// TIA Portal V18 export
// export: Created 2026-04-18T00:00:00Z, ExportSetting WithDefaults
ORGANIZATION_BLOCK "OB31_PID_PLC2_Bon4"   // OB31, LAD, CyclicInterrupt
{ S7_Optimized_Access := 'TRUE' }
VERSION : 0.1
// stored: AutoNumber true, IsIECCheckEnabled false
   VAR_INPUT
      Initial_Call : Bool;
      Remanence : Bool;
   END_VAR
BEGIN

REGION Network 1: Initialize PID Bon 4 Kp parameter
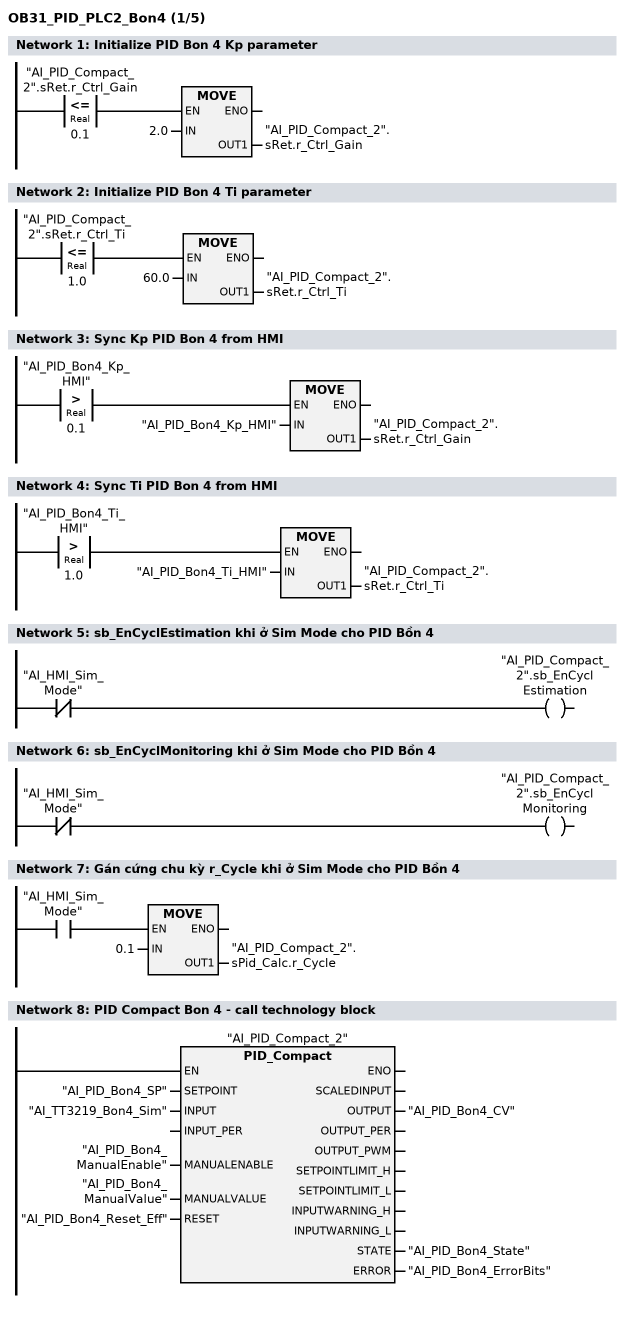
   RUNG wire#powerrail
      { S7_Templates := "SrcType := Real" } LE_Contact(in1 := "AI_PID_Compact_2".sRet.r_Ctrl_Gain, in2 := 0.1)
      { S7_GenerateENO := "TRUE" } Move(in := 2.0, out1 => "AI_PID_Compact_2".sRet.r_Ctrl_Gain)
   END_RUNG
   // the same network as SCL:
   IF "AI_PID_Compact_2".sRet.r_Ctrl_Gain <= 0.1 THEN "AI_PID_Compact_2".sRet.r_Ctrl_Gain := 2.0; END_IF;
END_REGION

REGION Network 2: Initialize PID Bon 4 Ti parameter
   RUNG wire#powerrail
      { S7_Templates := "SrcType := Real" } LE_Contact(in1 := "AI_PID_Compact_2".sRet.r_Ctrl_Ti, in2 := 1.0)
      { S7_GenerateENO := "TRUE" } Move(in := 60.0, out1 => "AI_PID_Compact_2".sRet.r_Ctrl_Ti)
   END_RUNG
   // the same network as SCL:
   IF "AI_PID_Compact_2".sRet.r_Ctrl_Ti <= 1.0 THEN "AI_PID_Compact_2".sRet.r_Ctrl_Ti := 60.0; END_IF;
END_REGION

REGION Network 3: Sync Kp PID Bon 4 from HMI
   RUNG wire#powerrail
      { S7_Templates := "SrcType := Real" } GT_Contact(in1 := "AI_PID_Bon4_Kp_HMI", in2 := 0.1)
      { S7_GenerateENO := "TRUE" } Move(in := "AI_PID_Bon4_Kp_HMI", out1 => "AI_PID_Compact_2".sRet.r_Ctrl_Gain)
   END_RUNG
   // the same network as SCL:
   IF "AI_PID_Bon4_Kp_HMI" > 0.1 THEN "AI_PID_Compact_2".sRet.r_Ctrl_Gain := "AI_PID_Bon4_Kp_HMI"; END_IF;
END_REGION

REGION Network 4: Sync Ti PID Bon 4 from HMI
   RUNG wire#powerrail
      { S7_Templates := "SrcType := Real" } GT_Contact(in1 := "AI_PID_Bon4_Ti_HMI", in2 := 1.0)
      { S7_GenerateENO := "TRUE" } Move(in := "AI_PID_Bon4_Ti_HMI", out1 => "AI_PID_Compact_2".sRet.r_Ctrl_Ti)
   END_RUNG
   // the same network as SCL:
   IF "AI_PID_Bon4_Ti_HMI" > 1.0 THEN "AI_PID_Compact_2".sRet.r_Ctrl_Ti := "AI_PID_Bon4_Ti_HMI"; END_IF;
END_REGION

REGION Network 5: sb_EnCyclEstimation khi ở Sim Mode cho PID Bồn 4
   RUNG wire#powerrail
      I_Contact( "AI_HMI_Sim_Mode" )
      Coil( "AI_PID_Compact_2".sb_EnCyclEstimation )
   END_RUNG
   // the same network as SCL:
   "AI_PID_Compact_2".sb_EnCyclEstimation := NOT "AI_HMI_Sim_Mode";
END_REGION

REGION Network 6: sb_EnCyclMonitoring khi ở Sim Mode cho PID Bồn 4
   RUNG wire#powerrail
      I_Contact( "AI_HMI_Sim_Mode" )
      Coil( "AI_PID_Compact_2".sb_EnCyclMonitoring )
   END_RUNG
   // the same network as SCL:
   "AI_PID_Compact_2".sb_EnCyclMonitoring := NOT "AI_HMI_Sim_Mode";
END_REGION

REGION Network 7: Gán cứng chu kỳ r_Cycle khi ở Sim Mode cho PID Bồn 4
   RUNG wire#powerrail
      Contact( "AI_HMI_Sim_Mode" )
      { S7_GenerateENO := "TRUE" } Move(in := 0.1, out1 => "AI_PID_Compact_2".sPid_Calc.r_Cycle)
   END_RUNG
   // the same network as SCL:
   IF "AI_HMI_Sim_Mode" THEN "AI_PID_Compact_2".sPid_Calc.r_Cycle := 0.1; END_IF;
END_REGION

REGION Network 8: PID Compact Bon 4 - call technology block
   RUNG wire#powerrail
      "AI_PID_Compact_2".PID_Compact(Setpoint := "AI_PID_Bon4_SP", Input := "AI_TT3219_Bon4_Sim", Input_PER :=, ManualEnable := "AI_PID_Bon4_ManualEnable", ManualValue := "AI_PID_Bon4_ManualValue", Reset := "AI_PID_Bon4_Reset_Eff", ScaledInput =>, Output => "AI_PID_Bon4_CV", Output_PER =>, Output_PWM =>, SetpointLimit_H =>, SetpointLimit_L =>, InputWarning_H =>, InputWarning_L =>, State => "AI_PID_Bon4_State", Error => "AI_PID_Bon4_ErrorBits")
   END_RUNG
   // the same network as SCL:
   "AI_PID_Compact_2"(Setpoint := "AI_PID_Bon4_SP",   // PID_Compact
                      Input := "AI_TT3219_Bon4_Sim",
                      ManualEnable := "AI_PID_Bon4_ManualEnable",
                      ManualValue := "AI_PID_Bon4_ManualValue",
                      Reset := "AI_PID_Bon4_Reset_Eff",
                      Output => "AI_PID_Bon4_CV",
                      State => "AI_PID_Bon4_State",
                      Error => "AI_PID_Bon4_ErrorBits");
END_REGION

REGION Network 9: Detect PID Bon 4 Error
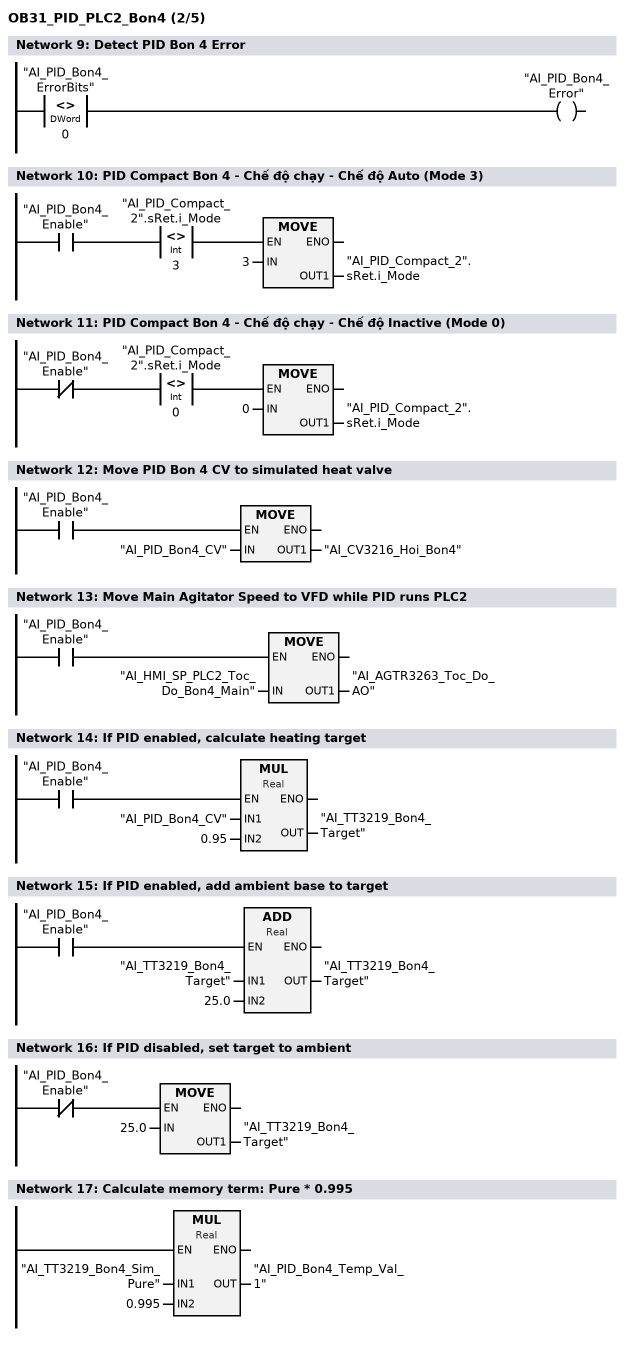
   RUNG wire#powerrail
      { S7_Templates := "SrcType := DWord" } NE_Contact(in1 := "AI_PID_Bon4_ErrorBits", in2 := 0)
      Coil( "AI_PID_Bon4_Error" )
   END_RUNG
   // the same network as SCL:
   "AI_PID_Bon4_Error" := "AI_PID_Bon4_ErrorBits" <> 0;
END_REGION

REGION Network 10: PID Compact Bon 4 - Chế độ chạy - Chế độ Auto (Mode 3)
   RUNG wire#powerrail
      Contact( "AI_PID_Bon4_Enable" )
      { S7_Templates := "SrcType := Int" } NE_Contact(in1 := "AI_PID_Compact_2".sRet.i_Mode, in2 := 3)
      { S7_GenerateENO := "TRUE" } Move(in := 3, out1 => "AI_PID_Compact_2".sRet.i_Mode)
   END_RUNG
   // the same network as SCL:
   IF "AI_PID_Bon4_Enable" AND ("AI_PID_Compact_2".sRet.i_Mode <> 3) THEN
       "AI_PID_Compact_2".sRet.i_Mode := 3;
   END_IF;
END_REGION

REGION Network 11: PID Compact Bon 4 - Chế độ chạy - Chế độ Inactive (Mode 0)
   RUNG wire#powerrail
      I_Contact( "AI_PID_Bon4_Enable" )
      { S7_Templates := "SrcType := Int" } NE_Contact(in1 := "AI_PID_Compact_2".sRet.i_Mode, in2 := 0)
      { S7_GenerateENO := "TRUE" } Move(in := 0, out1 => "AI_PID_Compact_2".sRet.i_Mode)
   END_RUNG
   // the same network as SCL:
   IF NOT "AI_PID_Bon4_Enable" AND ("AI_PID_Compact_2".sRet.i_Mode <> 0) THEN
       "AI_PID_Compact_2".sRet.i_Mode := 0;
   END_IF;
END_REGION

REGION Network 12: Move PID Bon 4 CV to simulated heat valve
   RUNG wire#powerrail
      Contact( "AI_PID_Bon4_Enable" )
      { S7_GenerateENO := "TRUE" } Move(in := "AI_PID_Bon4_CV", out1 => "AI_CV3216_Hoi_Bon4")
   END_RUNG
   // the same network as SCL:
   IF "AI_PID_Bon4_Enable" THEN "AI_CV3216_Hoi_Bon4" := "AI_PID_Bon4_CV"; END_IF;
END_REGION

REGION Network 13: Move Main Agitator Speed to VFD while PID runs PLC2
   RUNG wire#powerrail
      Contact( "AI_PID_Bon4_Enable" )
      { S7_GenerateENO := "TRUE" } Move(in := "AI_HMI_SP_PLC2_Toc_Do_Bon4_Main", out1 => "AI_AGTR3263_Toc_Do_AO")
   END_RUNG
   // the same network as SCL:
   IF "AI_PID_Bon4_Enable" THEN "AI_AGTR3263_Toc_Do_AO" := "AI_HMI_SP_PLC2_Toc_Do_Bon4_Main"; END_IF;
END_REGION

REGION Network 14: If PID enabled, calculate heating target
   RUNG wire#powerrail
      Contact( "AI_PID_Bon4_Enable" )
      { S7_Templates := "SrcType := Real"; S7_GenerateENO := "TRUE" } Mul(in1 := "AI_PID_Bon4_CV", in2 := 0.95, out => "AI_TT3219_Bon4_Target")
   END_RUNG
   // the same network as SCL:
   IF "AI_PID_Bon4_Enable" THEN "AI_TT3219_Bon4_Target" := "AI_PID_Bon4_CV" * 0.95; END_IF;
END_REGION

REGION Network 15: If PID enabled, add ambient base to target
   RUNG wire#powerrail
      Contact( "AI_PID_Bon4_Enable" )
      { S7_Templates := "SrcType := Real"; S7_GenerateENO := "TRUE" } Add(in1 := "AI_TT3219_Bon4_Target", in2 := 25.0, out => "AI_TT3219_Bon4_Target")
   END_RUNG
   // the same network as SCL:
   IF "AI_PID_Bon4_Enable" THEN "AI_TT3219_Bon4_Target" := "AI_TT3219_Bon4_Target" + 25.0; END_IF;
END_REGION

REGION Network 16: If PID disabled, set target to ambient
   RUNG wire#powerrail
      I_Contact( "AI_PID_Bon4_Enable" )
      { S7_GenerateENO := "TRUE" } Move(in := 25.0, out1 => "AI_TT3219_Bon4_Target")
   END_RUNG
   // the same network as SCL:
   IF NOT "AI_PID_Bon4_Enable" THEN "AI_TT3219_Bon4_Target" := 25.0; END_IF;
END_REGION

REGION Network 17: Calculate memory term: Pure * 0.995
   RUNG wire#powerrail
      { S7_Templates := "SrcType := Real"; S7_GenerateENO := "TRUE" } Mul(in1 := "AI_TT3219_Bon4_Sim_Pure", in2 := 0.995, out => "AI_PID_Bon4_Temp_Val_1")
   END_RUNG
   // the same network as SCL:
   "AI_PID_Bon4_Temp_Val_1" := "AI_TT3219_Bon4_Sim_Pure" * 0.995;
END_REGION

REGION Network 18: Calculate target term: Target * 0.005
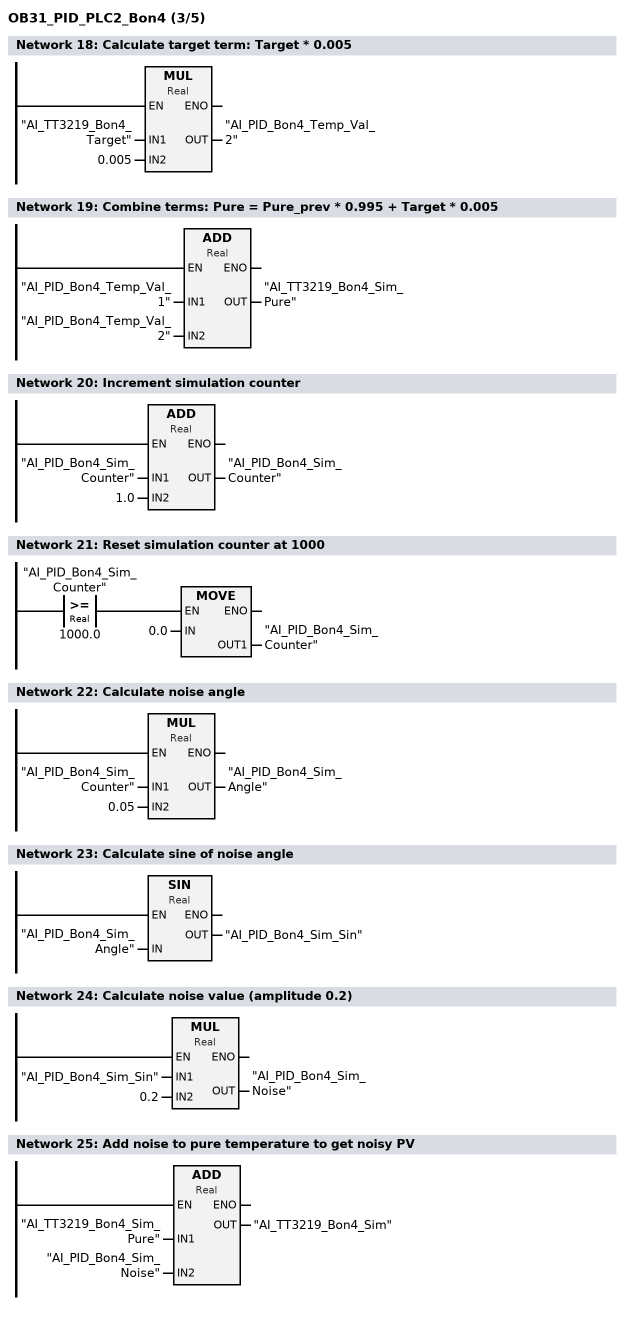
   RUNG wire#powerrail
      { S7_Templates := "SrcType := Real"; S7_GenerateENO := "TRUE" } Mul(in1 := "AI_TT3219_Bon4_Target", in2 := 0.005, out => "AI_PID_Bon4_Temp_Val_2")
   END_RUNG
   // the same network as SCL:
   "AI_PID_Bon4_Temp_Val_2" := "AI_TT3219_Bon4_Target" * 0.005;
END_REGION

REGION Network 19: Combine terms: Pure = Pure_prev * 0.995 + Target * 0.005
   RUNG wire#powerrail
      { S7_Templates := "SrcType := Real"; S7_GenerateENO := "TRUE" } Add(in1 := "AI_PID_Bon4_Temp_Val_1", in2 := "AI_PID_Bon4_Temp_Val_2", out => "AI_TT3219_Bon4_Sim_Pure")
   END_RUNG
   // the same network as SCL:
   "AI_TT3219_Bon4_Sim_Pure" := "AI_PID_Bon4_Temp_Val_1" + "AI_PID_Bon4_Temp_Val_2";
END_REGION

REGION Network 20: Increment simulation counter
   RUNG wire#powerrail
      { S7_Templates := "SrcType := Real"; S7_GenerateENO := "TRUE" } Add(in1 := "AI_PID_Bon4_Sim_Counter", in2 := 1.0, out => "AI_PID_Bon4_Sim_Counter")
   END_RUNG
   // the same network as SCL:
   "AI_PID_Bon4_Sim_Counter" := "AI_PID_Bon4_Sim_Counter" + 1.0;
END_REGION

REGION Network 21: Reset simulation counter at 1000
   RUNG wire#powerrail
      { S7_Templates := "SrcType := Real" } GE_Contact(in1 := "AI_PID_Bon4_Sim_Counter", in2 := 1000.0)
      { S7_GenerateENO := "TRUE" } Move(in := 0.0, out1 => "AI_PID_Bon4_Sim_Counter")
   END_RUNG
   // the same network as SCL:
   IF "AI_PID_Bon4_Sim_Counter" >= 1000.0 THEN "AI_PID_Bon4_Sim_Counter" := 0.0; END_IF;
END_REGION

REGION Network 22: Calculate noise angle
   RUNG wire#powerrail
      { S7_Templates := "SrcType := Real"; S7_GenerateENO := "TRUE" } Mul(in1 := "AI_PID_Bon4_Sim_Counter", in2 := 0.05, out => "AI_PID_Bon4_Sim_Angle")
   END_RUNG
   // the same network as SCL:
   "AI_PID_Bon4_Sim_Angle" := "AI_PID_Bon4_Sim_Counter" * 0.05;
END_REGION

REGION Network 23: Calculate sine of noise angle
   "AI_PID_Bon4_Sim_Sin" := SIN("AI_PID_Bon4_Sim_Angle");
END_REGION

REGION Network 24: Calculate noise value (amplitude 0.2)
   RUNG wire#powerrail
      { S7_Templates := "SrcType := Real"; S7_GenerateENO := "TRUE" } Mul(in1 := "AI_PID_Bon4_Sim_Sin", in2 := 0.2, out => "AI_PID_Bon4_Sim_Noise")
   END_RUNG
   // the same network as SCL:
   "AI_PID_Bon4_Sim_Noise" := "AI_PID_Bon4_Sim_Sin" * 0.2;
END_REGION

REGION Network 25: Add noise to pure temperature to get noisy PV
   RUNG wire#powerrail
      { S7_Templates := "SrcType := Real"; S7_GenerateENO := "TRUE" } Add(in1 := "AI_TT3219_Bon4_Sim_Pure", in2 := "AI_PID_Bon4_Sim_Noise", out => "AI_TT3219_Bon4_Sim")
   END_RUNG
   // the same network as SCL:
   "AI_TT3219_Bon4_Sim" := "AI_TT3219_Bon4_Sim_Pure" + "AI_PID_Bon4_Sim_Noise";
END_REGION

REGION Network 26: Đồng bộ giá trị mô phỏng sang tag HMI để truyền Modbus
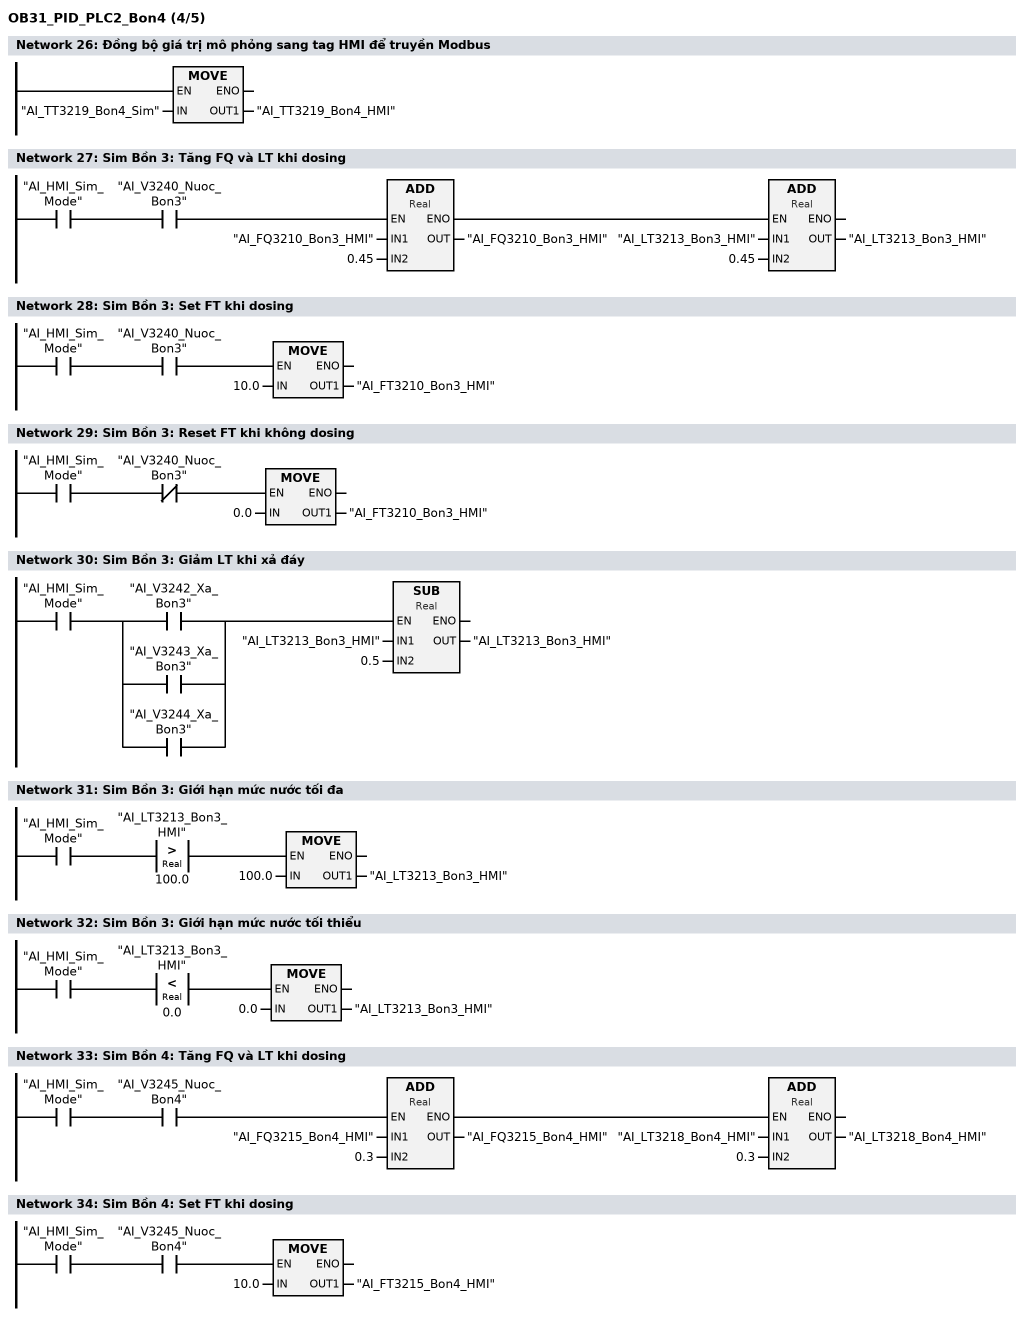
   RUNG wire#powerrail
      { S7_GenerateENO := "TRUE" } Move(in := "AI_TT3219_Bon4_Sim", out1 => "AI_TT3219_Bon4_HMI")
   END_RUNG
   // the same network as SCL:
   "AI_TT3219_Bon4_HMI" := "AI_TT3219_Bon4_Sim";
END_REGION

REGION Network 27: Sim Bồn 3: Tăng FQ và LT khi dosing
   RUNG wire#powerrail
      Contact( "AI_HMI_Sim_Mode" )
      Contact( "AI_V3240_Nuoc_Bon3" )
      { S7_Templates := "SrcType := Real"; S7_GenerateENO := "TRUE" } Add(in1 := "AI_FQ3210_Bon3_HMI", in2 := 0.45, out => "AI_FQ3210_Bon3_HMI")
      { S7_Templates := "SrcType := Real"; S7_GenerateENO := "TRUE" } Add(in1 := "AI_LT3213_Bon3_HMI", in2 := 0.45, out => "AI_LT3213_Bon3_HMI")
   END_RUNG
   // the same network as SCL:
   // ENO of a box is taken as its EN; it also drops when the box reports an error
   IF "AI_HMI_Sim_Mode" AND "AI_V3240_Nuoc_Bon3" THEN
       "AI_FQ3210_Bon3_HMI" := "AI_FQ3210_Bon3_HMI" + 0.45;
       "AI_LT3213_Bon3_HMI" := "AI_LT3213_Bon3_HMI" + 0.45;
   END_IF;
END_REGION

REGION Network 28: Sim Bồn 3: Set FT khi dosing
   RUNG wire#powerrail
      Contact( "AI_HMI_Sim_Mode" )
      Contact( "AI_V3240_Nuoc_Bon3" )
      { S7_GenerateENO := "TRUE" } Move(in := 10.0, out1 => "AI_FT3210_Bon3_HMI")
   END_RUNG
   // the same network as SCL:
   IF "AI_HMI_Sim_Mode" AND "AI_V3240_Nuoc_Bon3" THEN "AI_FT3210_Bon3_HMI" := 10.0; END_IF;
END_REGION

REGION Network 29: Sim Bồn 3: Reset FT khi không dosing
   RUNG wire#powerrail
      Contact( "AI_HMI_Sim_Mode" )
      I_Contact( "AI_V3240_Nuoc_Bon3" )
      { S7_GenerateENO := "TRUE" } Move(in := 0.0, out1 => "AI_FT3210_Bon3_HMI")
   END_RUNG
   // the same network as SCL:
   IF "AI_HMI_Sim_Mode" AND NOT "AI_V3240_Nuoc_Bon3" THEN "AI_FT3210_Bon3_HMI" := 0.0; END_IF;
END_REGION

REGION Network 30: Sim Bồn 3: Giảm LT khi xả đáy
   RUNG wire#powerrail
      Contact( "AI_HMI_Sim_Mode" )
      wire#w1
      Contact( "AI_V3242_Xa_Bon3" )
      wire#w2
      { S7_Templates := "SrcType := Real"; S7_GenerateENO := "TRUE" } Sub(in1 := "AI_LT3213_Bon3_HMI", in2 := 0.5, out => "AI_LT3213_Bon3_HMI")
   END_RUNG
   RUNG wire#w1
      Contact( "AI_V3243_Xa_Bon3" )
   END_RUNG wire#w2
   RUNG wire#w1
      Contact( "AI_V3244_Xa_Bon3" )
   END_RUNG wire#w2
   // the same network as SCL:
   IF "AI_HMI_Sim_Mode" AND ("AI_V3242_Xa_Bon3" OR "AI_V3243_Xa_Bon3" OR "AI_V3244_Xa_Bon3") THEN
       "AI_LT3213_Bon3_HMI" := "AI_LT3213_Bon3_HMI" - 0.5;
   END_IF;
END_REGION

REGION Network 31: Sim Bồn 3: Giới hạn mức nước tối đa
   RUNG wire#powerrail
      Contact( "AI_HMI_Sim_Mode" )
      { S7_Templates := "SrcType := Real" } GT_Contact(in1 := "AI_LT3213_Bon3_HMI", in2 := 100.0)
      { S7_GenerateENO := "TRUE" } Move(in := 100.0, out1 => "AI_LT3213_Bon3_HMI")
   END_RUNG
   // the same network as SCL:
   IF "AI_HMI_Sim_Mode" AND ("AI_LT3213_Bon3_HMI" > 100.0) THEN "AI_LT3213_Bon3_HMI" := 100.0; END_IF;
END_REGION

REGION Network 32: Sim Bồn 3: Giới hạn mức nước tối thiểu
   RUNG wire#powerrail
      Contact( "AI_HMI_Sim_Mode" )
      { S7_Templates := "SrcType := Real" } LT_Contact(in1 := "AI_LT3213_Bon3_HMI", in2 := 0.0)
      { S7_GenerateENO := "TRUE" } Move(in := 0.0, out1 => "AI_LT3213_Bon3_HMI")
   END_RUNG
   // the same network as SCL:
   IF "AI_HMI_Sim_Mode" AND ("AI_LT3213_Bon3_HMI" < 0.0) THEN "AI_LT3213_Bon3_HMI" := 0.0; END_IF;
END_REGION

REGION Network 33: Sim Bồn 4: Tăng FQ và LT khi dosing
   RUNG wire#powerrail
      Contact( "AI_HMI_Sim_Mode" )
      Contact( "AI_V3245_Nuoc_Bon4" )
      { S7_Templates := "SrcType := Real"; S7_GenerateENO := "TRUE" } Add(in1 := "AI_FQ3215_Bon4_HMI", in2 := 0.3, out => "AI_FQ3215_Bon4_HMI")
      { S7_Templates := "SrcType := Real"; S7_GenerateENO := "TRUE" } Add(in1 := "AI_LT3218_Bon4_HMI", in2 := 0.3, out => "AI_LT3218_Bon4_HMI")
   END_RUNG
   // the same network as SCL:
   // ENO of a box is taken as its EN; it also drops when the box reports an error
   IF "AI_HMI_Sim_Mode" AND "AI_V3245_Nuoc_Bon4" THEN
       "AI_FQ3215_Bon4_HMI" := "AI_FQ3215_Bon4_HMI" + 0.3;
       "AI_LT3218_Bon4_HMI" := "AI_LT3218_Bon4_HMI" + 0.3;
   END_IF;
END_REGION

REGION Network 34: Sim Bồn 4: Set FT khi dosing
   RUNG wire#powerrail
      Contact( "AI_HMI_Sim_Mode" )
      Contact( "AI_V3245_Nuoc_Bon4" )
      { S7_GenerateENO := "TRUE" } Move(in := 10.0, out1 => "AI_FT3215_Bon4_HMI")
   END_RUNG
   // the same network as SCL:
   IF "AI_HMI_Sim_Mode" AND "AI_V3245_Nuoc_Bon4" THEN "AI_FT3215_Bon4_HMI" := 10.0; END_IF;
END_REGION

REGION Network 35: Sim Bồn 4: Reset FT khi không dosing
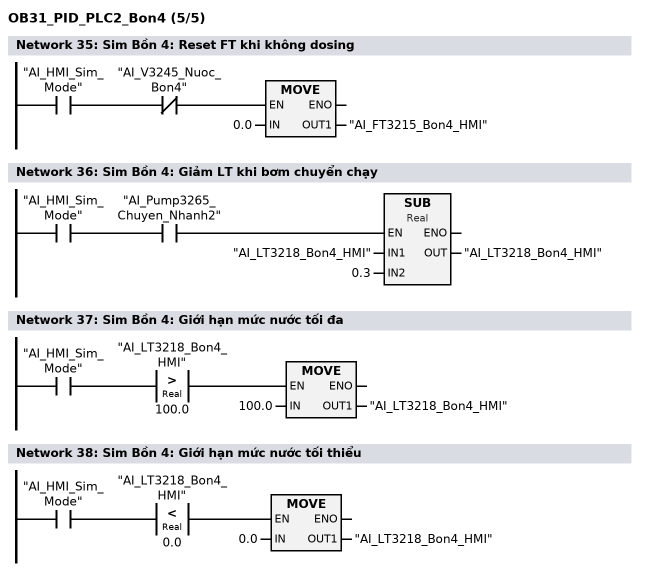
   RUNG wire#powerrail
      Contact( "AI_HMI_Sim_Mode" )
      I_Contact( "AI_V3245_Nuoc_Bon4" )
      { S7_GenerateENO := "TRUE" } Move(in := 0.0, out1 => "AI_FT3215_Bon4_HMI")
   END_RUNG
   // the same network as SCL:
   IF "AI_HMI_Sim_Mode" AND NOT "AI_V3245_Nuoc_Bon4" THEN "AI_FT3215_Bon4_HMI" := 0.0; END_IF;
END_REGION

REGION Network 36: Sim Bồn 4: Giảm LT khi bơm chuyển chạy
   RUNG wire#powerrail
      Contact( "AI_HMI_Sim_Mode" )
      Contact( "AI_Pump3265_Chuyen_Nhanh2" )
      { S7_Templates := "SrcType := Real"; S7_GenerateENO := "TRUE" } Sub(in1 := "AI_LT3218_Bon4_HMI", in2 := 0.3, out => "AI_LT3218_Bon4_HMI")
   END_RUNG
   // the same network as SCL:
   IF "AI_HMI_Sim_Mode" AND "AI_Pump3265_Chuyen_Nhanh2" THEN
       "AI_LT3218_Bon4_HMI" := "AI_LT3218_Bon4_HMI" - 0.3;
   END_IF;
END_REGION

REGION Network 37: Sim Bồn 4: Giới hạn mức nước tối đa
   RUNG wire#powerrail
      Contact( "AI_HMI_Sim_Mode" )
      { S7_Templates := "SrcType := Real" } GT_Contact(in1 := "AI_LT3218_Bon4_HMI", in2 := 100.0)
      { S7_GenerateENO := "TRUE" } Move(in := 100.0, out1 => "AI_LT3218_Bon4_HMI")
   END_RUNG
   // the same network as SCL:
   IF "AI_HMI_Sim_Mode" AND ("AI_LT3218_Bon4_HMI" > 100.0) THEN "AI_LT3218_Bon4_HMI" := 100.0; END_IF;
END_REGION

REGION Network 38: Sim Bồn 4: Giới hạn mức nước tối thiểu
   RUNG wire#powerrail
      Contact( "AI_HMI_Sim_Mode" )
      { S7_Templates := "SrcType := Real" } LT_Contact(in1 := "AI_LT3218_Bon4_HMI", in2 := 0.0)
      { S7_GenerateENO := "TRUE" } Move(in := 0.0, out1 => "AI_LT3218_Bon4_HMI")
   END_RUNG
   // the same network as SCL:
   IF "AI_HMI_Sim_Mode" AND ("AI_LT3218_Bon4_HMI" < 0.0) THEN "AI_LT3218_Bon4_HMI" := 0.0; END_IF;
END_REGION
END_ORGANIZATION_BLOCK
